(* CoDeSys 2.3 export: FX_PORTED.EXP *)

(* POU Simulation_Visuelle/FX_PorteD, ST *)
FUNCTION FX_PorteD : REAL
VAR_INPUT
	PosXPorte: INT;
END_VAR
VAR
	VarLocalA: REAL;
	ValXLocal: REAL;
END_VAR
(*Cette fonction retourne la position Y en fonction de l'axe X de la porte droite*)
VarLocalA:=(27.0/71.0);
ValXLocal:= INT_TO_REAL(PosXPorte);
VarLocalA:=(VarLocalA)*(ValXLocal);
FX_PorteD:=VarLocalA- 2;
END_FUNCTION
